{attribute 'TcGenerated'}
// This function has been automatically generated from the project information.
VAR_GLOBAL CONSTANT
	{attribute 'const_non_replaced'}
	{attribute 'linkalways'}
	stLibVersion_MBC_TC3_PCS_Library : ST_LibVersion := (iMajor := 1, iMinor := 1, iBuild := 0, iRevision := 0, sVersion := '1.1.0.0');
END_VAR

(* stored: Version 1.1.0.1, ProductVersion 3.1.4022.7
   GVL Global_Version: Id {b04f62c3-23a7-0bc4-3d46-52acd3064e70} *)
